// TIA Portal V16 export
// export: Created 2022-02-04T14:40:18.5433975Z, ExportSetting WithDefaults, DisplayName Totally Integrated Automation Portal, DisplayVersion V16 Update 1, DisplayName TIA Portal Version Control Interface, DisplayVersion V16, DisplayName TIA Portal Openness, DisplayVersion V16, DisplayName SINAMICS Startdrive Advanced, DisplayVersion V16 Update 5, DisplayName SINAMICS Startdrive G130, G150, S120, S150, SINAMICS MV, S210, DisplayVersion V16 Update 5, DisplayName SINAMICS Startdrive G110M, G120, G120C, G120D, G120P, G115D, DisplayVersion V16 Update 5, DisplayName STEP 7 Professional, DisplayVersion V16, DisplayName STEP 7 Safety, DisplayVersion V16, DisplayName WinCC Advanced, DisplayVersion V16, DisplayName SIMATIC Visualization Architect, DisplayVersion V16
DATA_BLOCK "Сортировка_DB"   // DB7
VERSION : 0.1
// stored: AutoNumber true, InstanceOfName Сортировка, InstanceOfType FB
"Сортировка"
   // VAR_INPUT
   //    packet_released : Bool;
   // END_VAR
   // VAR RETAIN
   //    "TrigE76.4" : Bool;
   //    Trig_Dovod : Bool;
   //    LiftPushingPacket : Bool;
   //    TrigAutoPFM : Bool;
   //    Trig_Vill : Bool;
   //    Trig_Vill2 : Bool;
   //    LiftDownTrig : Bool;
   //    HaveSxema : Bool;
   //    NewPacket : Bool;
   //    LiftDown_old : Bool;
   //    LiftPushing_old : Bool;
   //    ForksForcingFinish : Bool;
   //    LiftForcingFinish : Bool;
   //    CommonForcingPacket : Bool;
   //    ElevatorLowering : Bool;
   //    NoGasketMode : Bool;
   //    RampIsOn : Bool;
   //    RampIsOff : Bool;
   //    power_Vill : Bool;
   //    MakedLayer : Bool;
   //    AlarmLowerElevator : Bool;
   //    AlarmNotReadedPack : Bool;
   //    lift_return_trig : Bool;
   //    ramp_sync_old : Bool;
   //    BoardInLayerCounter : Int;
   //    LayersCounter : Int;
   //    Vibrator_KeyFazer { S7_SetPoint := 'True'} : "Vibrator";
   //    Run323_timer { S7_SetPoint := 'True'} : TP;
   //    LayerCounter { S7_SetPoint := 'True'} : "Adder";
   // END_VAR
BEGIN
END_DATA_BLOCK
